PROGRAM MAIN
VAR
	master 		: AXIS_REF;
	slave 		: AXIS_REF;
	fb_Power	: MC_Power;
	bEnable		: BOOL;
	fb_Power2	: MC_Power;
	fb_GearIn	: MC_GearIn;
	enable		: BOOL;
	fbMove 		: MC_MoveAbsolute;
	mEnable		: BOOL;
	fb_GearOut	: MC_GearOut;
	nenable		: BOOL;
	fb_Stop		: MC_Stop;
	fb_halt 	:MC_Halt;
	bStop 		: BOOL:=FALSE;
	deger 		: LREAL;

	d: BOOL;
	dEnable: BOOL;
END_VAR


fb_Power(//For master
	Axis:=master , 
	Enable:= bEnable, 
	Enable_Positive:= bEnable, 
	Enable_Negative:= bEnable, 
	Override:=100 );
	
fb_Power2(//for slave
	Axis:=slave , 
	Enable:=bEnable , 
	Enable_Positive:=bEnable , 
	Enable_Negative:= bEnable, 
	Override:=100 );
	

fb_GearIn(
	Master:=master , 
	Slave:= slave, 
	Execute:= enable, 
	RatioNumerator:=5 , 
	RatioDenominator:= 1);
	
fbMove(
	Axis:=master , 
	Execute:=mEnable , 
	Position:=deger , 
	Velocity:= 100 );
	
	
fb_GearOut(
	Slave:= slave, 
	Execute:=nenable);
	
fb_Stop(
	Axis:= master, 
	Execute:=bStop);
	

fb_halt(
	Axis:=master , 
	Execute:= dEnable);

END_PROGRAM

(* stored: Version 1.1.0.1, ProductVersion 3.1.4024.12
   POU MAIN: Id {52817031-2ae7-47a1-964d-2a226199c577}, SpecialFunc None *)
